# EPICS StreamDevice protocol: demopIOC/protocols/NEWFOCUS8742.proto
OutTerminator = CR;
InTerminator = CR LF;
getIPAddress
{
	out "IPADDR?";
	in "%s";
}
move_relative
{
	out "%(\$1)iPR%i";
}
getVELO
{
	out "%(\$1)iVA?";
	in "%i";
}
SetVelo
{
	out "%(\$1)iVA%i";
}
